# EPICS substitutions: BLDApp/Db/BLDMCastReceiverGdets.substitutions
file BLDMCastReceiverGdet.template
{
#         Station			MC Group	Stat_Scan
pattern { STN			,	MC,			STAT_SCAN	}
        { "FEEGasDetEnergy"	,  	"2"			"5"	}
}
